# EPICS substitutions: alsuPSC_4Channel_skew/pscApp/Db/BipPkt.substitutions
file BipPkt.template
{pattern
{BYTENUM,REG,WORDNUM}
#Bipolar Packet 1
{144 ,0 ,1}
{148 ,1 ,1}
{152 ,2 ,1}
{156 ,3 ,1}
{160 ,4 ,1}
{164 ,5 ,1}
{168 ,6 ,1}
{172 ,7 ,1}
{176 ,8 ,1}
{180 ,9 ,1}
{184 ,10,1}
{188 ,11,1}
{192 ,12,1}
{196 ,13,1}
{200 ,14,1}
{204 ,15,1}
{208 ,16,1}
{212 ,17,1}
{216 ,18,1}
{220 ,19,1}
{224 ,20,1}
{228 ,21,1}
{232 ,22,1}
{236 ,23,1}
{240 ,24,1}
{244 ,25,1}
{248 ,26,1}
{252 ,27,1}
{256 ,28,1}
{260 ,29,1}
{264 ,30,1}
{268 ,31,1}
{272 ,32,1}
{276 ,33,1}
{280 ,34,1}
{284 ,35,1}
{288 ,36,1}
{292 ,37,1}
{296 ,38,1}
{300 ,39,1}
{304 ,40,1}
{308 ,41,1}
{312 ,42,1}
{316 ,43,1}
{320 ,44,1}
{324 ,45,1}
{328 ,46,1}
{332 ,47,1}
{336 ,48,1}
{340 ,49,1}
{344 ,50,1}
{348 ,51,1}
{352 ,52,1}
{356 ,53,1}
{360 ,54,1}
{364 ,55,1}
{368 ,56,1}
{372 ,57,1}
{376 ,58,1}
{380 ,59,1}
#Bipolar Packet 2
{384 ,0 ,2}
{388 ,1 ,2}
{392 ,2 ,2}
{396 ,3 ,2}
{400 ,4 ,2}
{404 ,5 ,2}
{408 ,6 ,2}
{412 ,7 ,2}
{416 ,8 ,2}
{420 ,9 ,2}
{424 ,10,2}
{428 ,11,2}
{432 ,12,2}
{436 ,13,2}
{440 ,14,2}
{444 ,15,2}
{448 ,16,2}
{452 ,17,2}
{456 ,18,2}
{460 ,19,2}
{464 ,20,2}
{468 ,21,2}
{472 ,22,2}
{476 ,23,2}
{480 ,24,2}
{484 ,25,2}
{488 ,26,2}
{492 ,27,2}
{496 ,28,2}
{500 ,29,2}
{504 ,30,2}
{508 ,31,2}
{512 ,32,2}
{516 ,33,2}
{520 ,34,2}
{524 ,35,2}
{528 ,36,2}
{532 ,37,2}
{536 ,38,2}
{540 ,39,2}
{544 ,40,2}
{548 ,41,2}
{552 ,42,2}
{556 ,43,2}
{560 ,44,2}
{564 ,45,2}
{568 ,46,2}
{572 ,47,2}
{576 ,48,2}
{580 ,49,2}
{584 ,50,2}
{588 ,51,2}
{592 ,52,2}
{596 ,53,2}
{600 ,54,2}
{604 ,55,2}
{608 ,56,2}
{612 ,57,2}
{616 ,58,2}
{620 ,59,2}
#Bipolar Packet 3
{624 ,0 ,3}
{628 ,1 ,3}
{632 ,2 ,3}
{636 ,3 ,3}
{640 ,4 ,3}
{644 ,5 ,3}
{648 ,6 ,3}
{652 ,7 ,3}
{656 ,8 ,3}
{660 ,9 ,3}
{664 ,10,3}
{668 ,11,3}
{672 ,12,3}
{676 ,13,3}
{680 ,14,3}
{684 ,15,3}
{688 ,16,3}
{692 ,17,3}
{696 ,18,3}
{700 ,19,3}
{704 ,20,3}
{708 ,21,3}
{712 ,22,3}
{716 ,23,3}
{720 ,24,3}
{724 ,25,3}
{728 ,26,3}
{732 ,27,3}
{736 ,28,3}
{740 ,29,3}
{744 ,30,3}
{748 ,31,3}
{752 ,32,3}
{756 ,33,3}
{760 ,34,3}
{764 ,35,3}
{768 ,36,3}
{772 ,37,3}
{776 ,38,3}
{780 ,39,3}
{784 ,40,3}
{788 ,41,3}
{792 ,42,3}
{796 ,43,3}
{800 ,44,3}
{804 ,45,3}
{808 ,46,3}
{812 ,47,3}
{816 ,48,3}
{820 ,49,3}
{824 ,50,3}
{828 ,51,3}
{832 ,52,3}
{836 ,53,3}
{840 ,54,3}
{844 ,55,3}
{848 ,56,3}
{852 ,57,3}
{856 ,58,3}
{860 ,59,3}
#Bipolar Packet 4
{864 ,0 ,4}
{868 ,1 ,4}
{872 ,2 ,4}
{876 ,3 ,4}
{880 ,4 ,4}
{884 ,5 ,4}
{888 ,6 ,4}
{892 ,7 ,4}
{896 ,8 ,4}
{900 ,9 ,4}
{904 ,10,4}
{908 ,11,4}
{912 ,12,4}
{916 ,13,4}
{920 ,14,4}
{924 ,15,4}
{928 ,16,4}
{932 ,17,4}
{936 ,18,4}
{940 ,19,4}
{944 ,20,4}
{948 ,21,4}
{952 ,22,4}
{956 ,23,4}
{960 ,24,4}
{964 ,25,4}
{968 ,26,4}
{972 ,27,4}
{976 ,28,4}
{980 ,29,4}
{984 ,30,4}
{988 ,31,4}
{992 ,32,4}
{996 ,33,4}
{1000,34,4}
{1004,35,4}
{1008,36,4}
{1012,37,4}
{1016,38,4}
{1020,39,4}
{1024,40,4}
{1028,41,4}
{1032,42,4}
{1036,43,4}
{1040,44,4}
{1044,45,4}
{1048,46,4}
{1052,47,4}
{1056,48,4}
{1060,49,4}
{1064,50,4}
{1068,51,4}
{1072,52,4}
{1076,53,4}
{1080,54,4}
{1084,55,4}
{1088,56,4}
{1092,57,4}
{1096,58,4}
{1100,59,4}

#NOTE:
#Started at 144 + (4*240) = 1104
#For Status Packet the position
#in the packet is the position -4 bytes so 1104 bytes - 4 bytes = 1100
}
